(* CoDeSys 2.3 export: FB_PIDCNTRL.EXP *)

(* POU new FB:s/FB_PIDcntrl, FBD *)
(*
FB to control actuator using analog input as feedback for pid controller. Output is pwm.

PID2:
The manipulated variable Y is already standardised to PWM1000
TUNING:
Select TN according to the time characteristics of the system: fast system = small TN slow system = large TN
. Slowly increment KP gradually, up to a value at which still definitely no fluctuation will occur.
. Readjust TN if necessary.
. Add differential component only if necessary: Select a TV value approx. 2...10 times smaller than TN. Select a KD value more or less similar to KP.
Note that the maximum control deviation is + 127. For good control characteristics this range should not be exceeded, but it should be exploited to the best possible extent
Parameter			 Data type 					Description
X					 WORD					input value
XS					 WORD					preset value
XMAX				 WORD					maximum preset value
KP					 REAL						Proportional component of the output signal (only positive values permissible)
KI					 REAL						Integral component of the output signal (only positive values permissible)
TN					 TIME						integral action time (integral component)
KD					 REAL						Differential component of the output signal (only positive values permissible)
TV					 TIME						derivative action time (differential component)
RESET			 BOOL						TRUE: reset the function element
												FALSE: function element is not executed.
Y					WORD						Manipulated variable(0..1000‰)

INPUT_ANALOGUE:
MODE(DEC)			Input operating mode						Global variable				FB OUT				UNIT
0						deactivated								IN_NOMODE					
1						binary input, minus switching (BH)		IN_DIGITAL_H					0 / 1
2						binary input, plus switching (BL)			IN_DIGITAL_L					0 / 1
4						current input								IN_CURRENT					0…20 000				µA				
8						voltage input								IN_VOLTAGE10				0…10 000				mV		
16						voltage input								IN_VOLTAGE30				0…32 000				mV		
32						voltage input, ratiometric					IN_RATIO						0…1 000				‰								
64
128
256
512					resistance input							IN_RESISTANCE				3...680					Ohm
																									16...30 000
PWM1000:
INIT : BOOL;						(* To initialize it *)
FREQUENCY : WORD;			(* PWM frequency in Hz *)
CHANNEL : BYTE;				(* 0 .. 15 *)
VALUE : WORD;					(* Duty cycle in permille *)
CHANGE : BOOL;					(* To change the frequency, duty cycle or dither value *)
DITHER_VALUE : WORD;			(* Dither value in permille *)
DITHER_FREQUENCY : WORD;	(* Dither frequency in Hz *)
	
*)					

FUNCTION_BLOCK FB_PIDcntrl
VAR_INPUT
	_uitemperatureSensorValue					:UINT;
	_itemperatureSP								:INT;
	_xenableChannel								:BOOL;
	_imode										:INT;
	_byInChannel									:BYTE;
	_rlinearInMin									:REAL;
	_rlinearInMax									:REAL;
	_rlinearOutMin								:REAL;
	_rlinearOutMax								:REAL;
	_byOutPwnChannel							:BYTE;
	_xinitPwm										:BOOL;
	_ipwmFreq									:INT;
	_pwmChange									:BOOL;
	_uipwmdither									:UINT;
	_uipwmdithefreq								:UINT;
	_rKP											:REAL;
	_rKI											:REAL;
	_tTN											:TIME;
	_rKD											:REAL;
	_tTV											:TIME;


END_VAR
VAR_OUTPUT
END_VAR
VAR
	_fbpid											:PID2;
	_fbpwm										:PWM1000;
	_fblinearscale									:LIN_TRAFO;
	_fbinanalog									:INPUT_ANALOG;
	_ixmaxpid										:INT;
	_xpidreset										:BOOL;

END_VAR
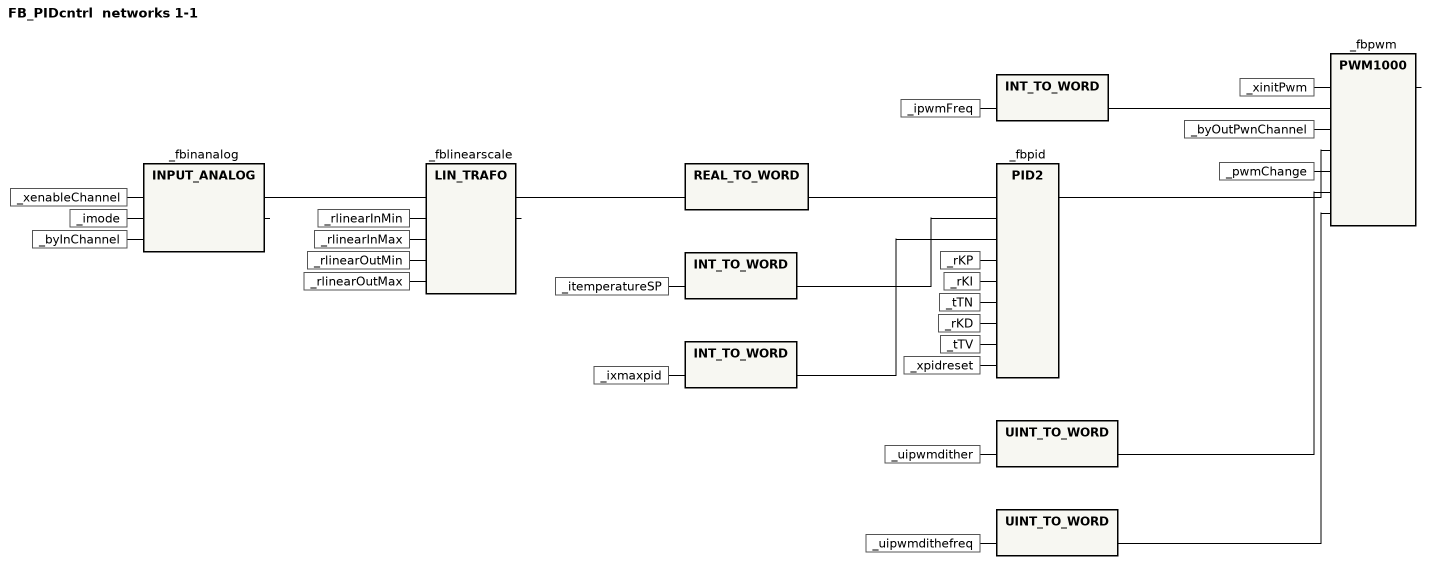
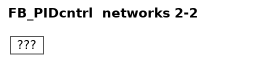
_FBD_ (* Function Block Diagram *)
NETWORK 1
	_fbpwm:PWM1000(_xinitPwm, INT_TO_WORD(_ipwmFreq), _byOutPwnChannel, _fbpid:PID2(REAL_TO_WORD(_fblinearscale:LIN_TRAFO(_fbinanalog:INPUT_ANALOG(_xenableChannel, _imode, _byInChannel), _rlinearInMin, _rlinearInMax, _rlinearOutMin, _rlinearOutMax)), INT_TO_WORD(_itemperatureSP), INT_TO_WORD(_ixmaxpid), _rKP, _rKI, _tTN, _rKD, _tTV, _xpidreset), _pwmChange, UINT_TO_WORD(_uipwmdither), UINT_TO_WORD(_uipwmdithefreq))
NETWORK 2
	???
_END_FBD_
END_FUNCTION_BLOCK
